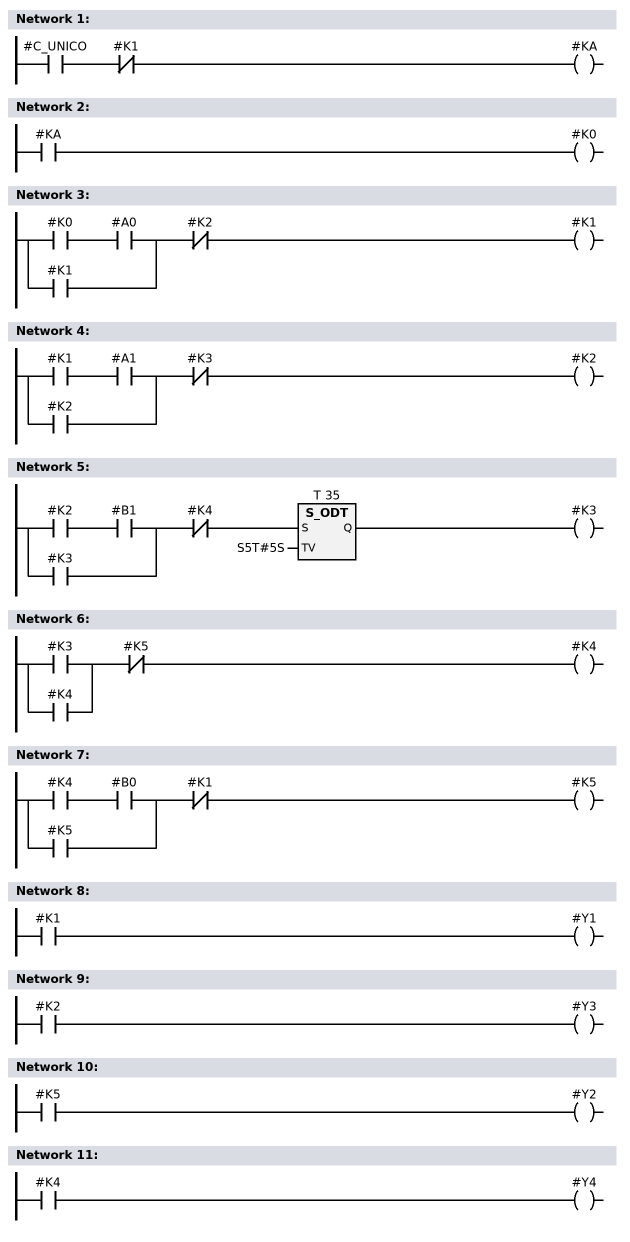
NETWORK
TITLE =
      A     #C_UNICO;
      AN    #K1;
      =     #KA;
NETWORK
TITLE =
      A     #KA;
      =     #K0;
NETWORK
TITLE =
      A(;
      A     #K0;
      A     #A0;
      O     #K1;
      );
      AN    #K2;
      =     #K1;
NETWORK
TITLE =
      A(;
      A     #K1;
      A     #A1;
      O     #K2;
      );
      AN    #K3;
      =     #K2;
NETWORK
TITLE =
      A(;
      A     #K2;
      A     #B1;
      O     #K3;
      );
      AN    #K4;
      L     S5T#5S;
      SD    T 35;
      NOP   0;
      NOP   0;
      NOP   0;
      A     T 35;
      =     #K3;
NETWORK
TITLE =
      A(;
      O     #K3;
      O     #K4;
      );
      AN    #K5;
      =     #K4;
NETWORK
TITLE =
      A(;
      A     #K4;
      A     #B0;
      O     #K5;
      );
      AN    #K1;
      =     #K5;
NETWORK
TITLE =
      A     #K1;
      =     #Y1;
NETWORK
TITLE =
      A     #K2;
      =     #Y3;
NETWORK
TITLE =
      A     #K5;
      =     #Y2;
NETWORK
TITLE =
      A     #K4;
      =     #Y4;
END_FUNCTION_BLOCK

FUNCTION_BLOCK "Ejercicio 6-3"	// FB 14
VERSION : 0.1
VAR_INPUT
  HONGO : BOOL ;
  RESET : BOOL ;
  C_UNICO : BOOL ;
  C_CONTINUO : BOOL ;
  PARO : BOOL ;
  DET_PIEZA : BOOL ;
  A0 : BOOL ;
  A1 : BOOL ;
  B0 : BOOL ;
  B1 : BOOL ;
  C0 : BOOL ;
  C1 : BOOL ;
END_VAR
VAR_OUTPUT
  Y1 : BOOL ;
  Y2 : BOOL ;
  Y3 : BOOL ;
  Y4 : BOOL ;
  Y5 : BOOL ;
  Y6 : BOOL ;
END_VAR
VAR
  K_PEM : BOOL ;
  KA : BOOL ;
  KB : BOOL ;
  K0 : BOOL ;
  K1 : BOOL ;
  K2 : BOOL ;
  K3 : BOOL ;
  K4 : BOOL ;
  K5 : BOOL ;
  K6 : BOOL ;
  K7 : BOOL ;
  K8 : BOOL ;
END_VAR
BEGIN
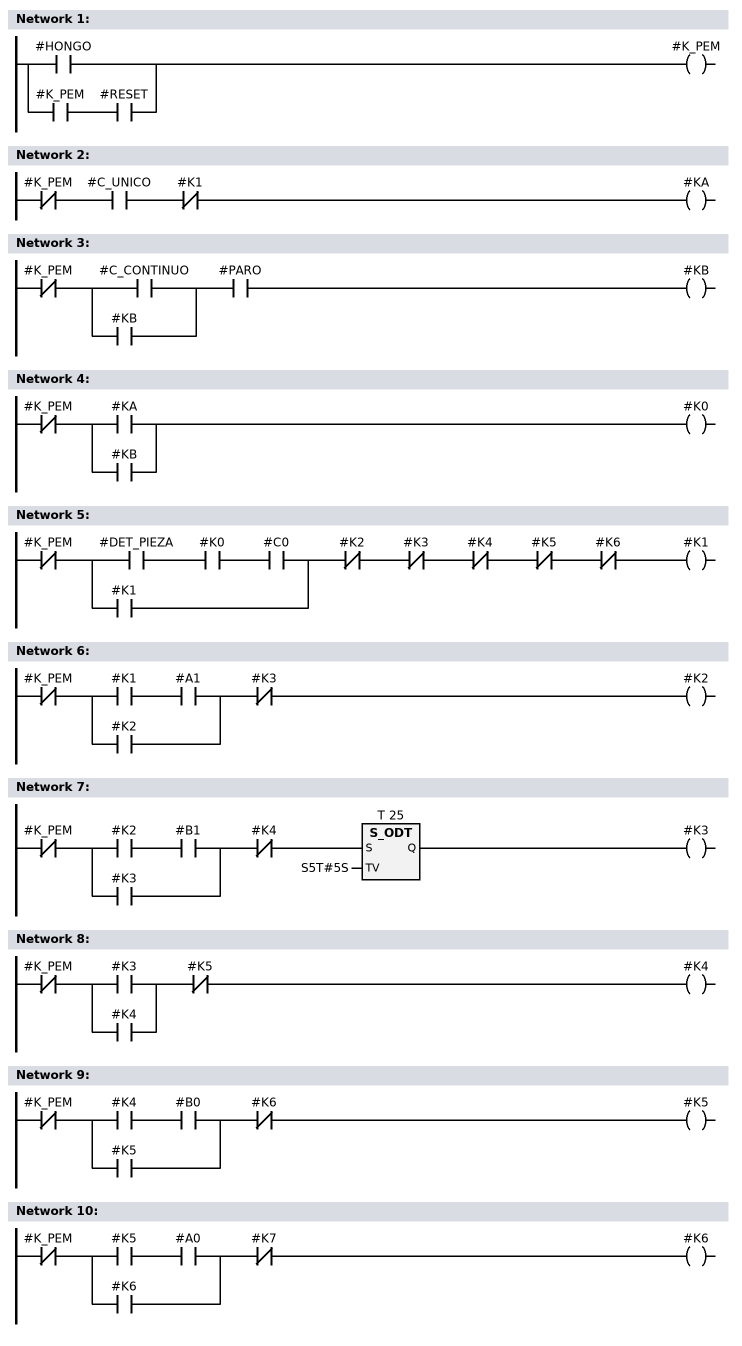
NETWORK
TITLE =
      O     #HONGO;
      O;
      A     #K_PEM;
      A     #RESET;
      =     #K_PEM;
NETWORK
TITLE =
      AN    #K_PEM;
      A     #C_UNICO;
      AN    #K1;
      =     #KA;
NETWORK
TITLE =
      AN    #K_PEM;
      A(;
      O     #C_CONTINUO;
      O     #KB;
      );
      A     #PARO;
      =     #KB;
NETWORK
TITLE =
      AN    #K_PEM;
      A(;
      O     #KA;
      O     #KB;
      );
      =     #K0;
NETWORK
TITLE =
      AN    #K_PEM;
      A(;
      A     #DET_PIEZA;
      A     #K0;
      A     #C0;
      O     #K1;
      );
      AN    #K2;
      AN    #K3;
      AN    #K4;
      AN    #K5;
      AN    #K6;
      =     #K1;
NETWORK
TITLE =
      AN    #K_PEM;
      A(;
      A     #K1;
      A     #A1;
      O     #K2;
      );
      AN    #K3;
      =     #K2;
NETWORK
TITLE =
      AN    #K_PEM;
      A(;
      A     #K2;
      A     #B1;
      O     #K3;
      );
      AN    #K4;
      L     S5T#5S;
      SD    T 25;
      NOP   0;
      NOP   0;
      NOP   0;
      A     T 25;
      =     #K3;
NETWORK
TITLE =
      AN    #K_PEM;
      A(;
      O     #K3;
      O     #K4;
      );
      AN    #K5;
      =     #K4;
NETWORK
TITLE =
      AN    #K_PEM;
      A(;
      A     #K4;
      A     #B0;
      O     #K5;
      );
      AN    #K6;
      =     #K5;
NETWORK
TITLE =
      AN    #K_PEM;
      A(;
      A     #K5;
      A     #A0;
      O     #K6;
      );
      AN    #K7;
      =     #K6;
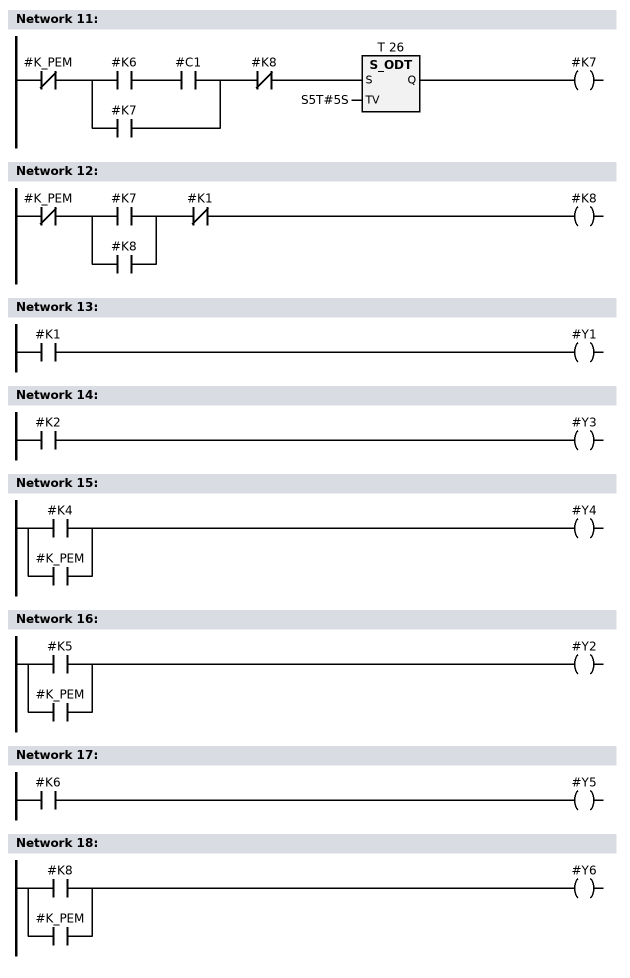
NETWORK
TITLE =
      AN    #K_PEM;
      A(;
      A     #K6;
      A     #C1;
      O     #K7;
      );
      AN    #K8;
      L     S5T#5S;
      SD    T 26;
      NOP   0;
      NOP   0;
      NOP   0;
      A     T 26;
      =     #K7;
NETWORK
TITLE =
      AN    #K_PEM;
      A(;
      O     #K7;
      O     #K8;
      );
      AN    #K1;
      =     #K8;
NETWORK
TITLE =
      A     #K1;
      =     #Y1;
NETWORK
TITLE =
      A     #K2;
      =     #Y3;
NETWORK
TITLE =
      O     #K4;
      O     #K_PEM;
      =     #Y4;
NETWORK
TITLE =
      O     #K5;
      O     #K_PEM;
      =     #Y2;
NETWORK
TITLE =
      A     #K6;
      =     #Y5;
NETWORK
TITLE =
      O     #K8;
      O     #K_PEM;
      =     #Y6;
END_FUNCTION_BLOCK

FUNCTION_BLOCK "Paro de emergencia"	// FB 99
VERSION : 0.1
VAR_INPUT
  HONGO : BOOL ;
  RESET : BOOL ;
END_VAR
VAR_OUTPUT
  K_PEM : BOOL ;
END_VAR
BEGIN
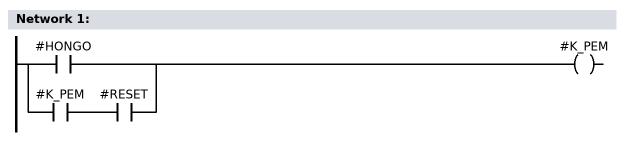
NETWORK
TITLE =
      O     #HONGO;
      O;
      A     #K_PEM;
      A     #RESET;
      =     #K_PEM;
END_FUNCTION_BLOCK

DATA_BLOCK DB 1
VERSION : 0.0
"Ejercicio1"
BEGIN
END_DATA_BLOCK

DATA_BLOCK DB 2
VERSION : 0.0
"Ejercicio 2"
BEGIN
END_DATA_BLOCK

DATA_BLOCK DB 3
VERSION : 0.0
"Ejercicio3"
BEGIN
END_DATA_BLOCK

DATA_BLOCK DB 4
VERSION : 0.0
"Ejercicio 4"
BEGIN
END_DATA_BLOCK

DATA_BLOCK DB 5
VERSION : 0.0
"Ejercicio 5"
BEGIN
END_DATA_BLOCK

DATA_BLOCK DB 6
VERSION : 0.0
"Ejercicio 6"
BEGIN
END_DATA_BLOCK

DATA_BLOCK DB 7
VERSION : 0.0
"Ejercicio C1"
BEGIN
END_DATA_BLOCK

DATA_BLOCK DB 8
VERSION : 0.0
"Ejercicio C2"
BEGIN
END_DATA_BLOCK

DATA_BLOCK DB 9
VERSION : 0.0
"Ejercicio 3-5"
BEGIN
END_DATA_BLOCK

DATA_BLOCK DB 10
VERSION : 0.0
"Ejercicio 3-6"
BEGIN
END_DATA_BLOCK

DATA_BLOCK DB 11
VERSION : 0.0
"Ejercicio 3-7"
BEGIN
END_DATA_BLOCK

DATA_BLOCK DB 12
VERSION : 0.0
"Ejercicio 6-1"
BEGIN
END_DATA_BLOCK

DATA_BLOCK DB 13
VERSION : 0.0
"Ejercicio 6-2"
BEGIN
END_DATA_BLOCK

DATA_BLOCK DB 14
VERSION : 0.0
"Ejercicio 6-3"
BEGIN
END_DATA_BLOCK

DATA_BLOCK DB 88
VERSION : 0.0
"Paro de emergencia"
BEGIN
END_DATA_BLOCK

DATA_BLOCK DB 89
VERSION : 0.0
"Paro de emergencia"
BEGIN
END_DATA_BLOCK

DATA_BLOCK DB 90
VERSION : 0.0
"Paro de emergencia"
BEGIN
END_DATA_BLOCK

DATA_BLOCK DB 91
VERSION : 0.0
"Paro de emergencia"
BEGIN
END_DATA_BLOCK

DATA_BLOCK DB 92
VERSION : 0.0
"Paro de emergencia"
BEGIN
END_DATA_BLOCK

DATA_BLOCK DB 93
VERSION : 0.0
"Paro de emergencia"
BEGIN
END_DATA_BLOCK

DATA_BLOCK DB 94
VERSION : 0.0
"Paro de emergencia"
BEGIN
END_DATA_BLOCK

DATA_BLOCK DB 95
VERSION : 0.0
"Paro de emergencia"
BEGIN
END_DATA_BLOCK

DATA_BLOCK DB 96
VERSION : 0.0
"Paro de emergencia"
BEGIN
END_DATA_BLOCK

DATA_BLOCK DB 97
VERSION : 0.0
"Paro de emergencia"
BEGIN
END_DATA_BLOCK

DATA_BLOCK DB 98
VERSION : 0.0
"Paro de emergencia"
BEGIN
END_DATA_BLOCK

DATA_BLOCK DB 99
VERSION : 0.0
"Paro de emergencia"
BEGIN
END_DATA_BLOCK

ORGANIZATION_BLOCK "CYCL_EXC"	// OB 1
TITLE = "Main Program Sweep (Cycle)"
VERSION : 0.1
VAR_TEMP
  OB1_EV_CLASS : BYTE ;	//Bits 0-3 = 1 (Coming event), Bits 4-7 = 1 (Event class 1)
  OB1_SCAN_1 : BYTE ;	//1 (Cold restart scan 1 of OB 1), 3 (Scan 2-n of OB 1)
  OB1_PRIORITY : BYTE ;	//Priority of OB Execution
  OB1_OB_NUMBR : BYTE ;	//1 (Organization block 1, OB1)
  OB1_RESERVED_1 : BYTE ;	//Reserved for system
  OB1_RESERVED_2 : BYTE ;	//Reserved for system
  OB1_PREV_CYCLE : INT ;	//Cycle time of previous OB1 scan (milliseconds)
  OB1_MIN_CYCLE : INT ;	//Minimum cycle time of OB1 (milliseconds)
  OB1_MAX_CYCLE : INT ;	//Maximum cycle time of OB1 (milliseconds)
  OB1_DATE_TIME : DATE_AND_TIME ;	//Date and time OB1 started
END_VAR
BEGIN
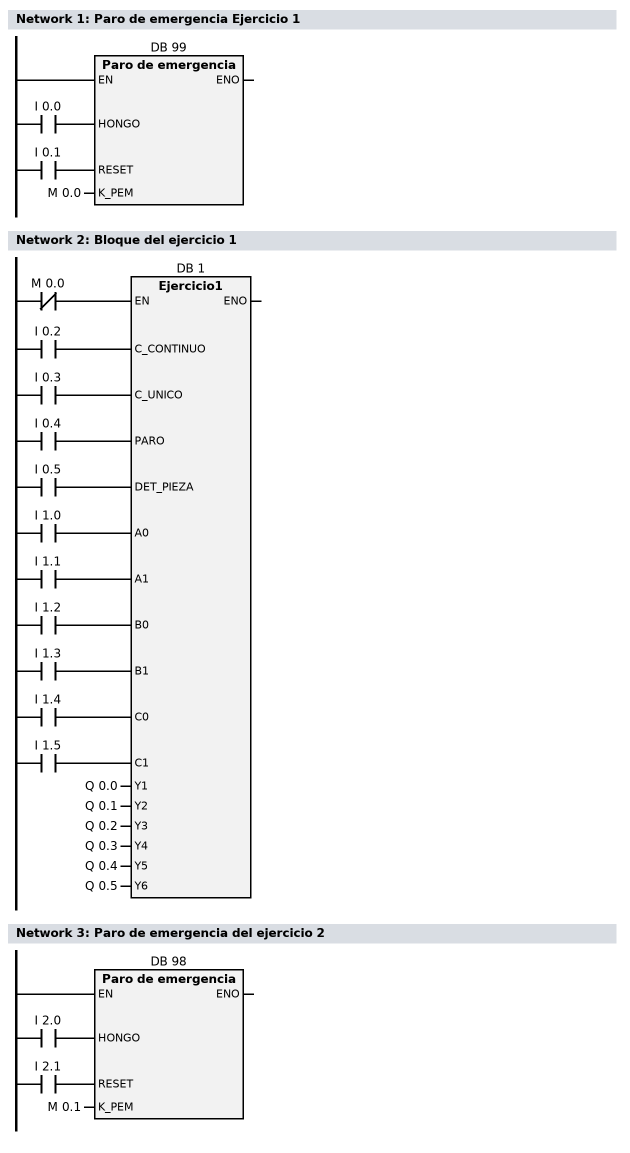
NETWORK
TITLE = Paro de emergencia Ejercicio 1
      A     I 0.0;
      =     L 20.0;
      BLD   103;
      A     I 0.1;
      =     L 20.1;
      BLD   103;
      CALL  "Paro de emergencia" , DB 99 (
           HONGO                    := L 20.0,
           RESET                    := L 20.1,
           K_PEM                    := M 0.0);
      NOP   0;
NETWORK
TITLE = Bloque del ejercicio 1
      A     I 0.2;
      =     L 20.0;
      BLD   103;
      A     I 0.3;
      =     L 20.1;
      BLD   103;
      A     I 0.4;
      =     L 20.2;
      BLD   103;
      A     I 0.5;
      =     L 20.3;
      BLD   103;
      A     I 1.0;
      =     L 20.4;
      BLD   103;
      A     I 1.1;
      =     L 20.5;
      BLD   103;
      A     I 1.2;
      =     L 20.6;
      BLD   103;
      A     I 1.3;
      =     L 20.7;
      BLD   103;
      A     I 1.4;
      =     L 21.0;
      BLD   103;
      A     I 1.5;
      =     L 21.1;
      BLD   103;
      AN    M 0.0;
      JNB   _001;
      CALL  "Ejercicio1" , DB 1 (
           C_CONTINUO               := L 20.0,
           C_UNICO                  := L 20.1,
           PARO                     := L 20.2,
           DET_PIEZA                := L 20.3,
           A0                       := L 20.4,
           A1                       := L 20.5,
           B0                       := L 20.6,
           B1                       := L 20.7,
           C0                       := L 21.0,
           C1                       := L 21.1,
           Y1                       := Q 0.0,
           Y2                       := Q 0.1,
           Y3                       := Q 0.2,
           Y4                       := Q 0.3,
           Y5                       := Q 0.4,
           Y6                       := Q 0.5);
_001: NOP   0;
NETWORK
TITLE = Paro de emergencia del ejercicio 2
      A     I 2.0;
      =     L 20.0;
      BLD   103;
      A     I 2.1;
      =     L 20.1;
      BLD   103;
      CALL  "Paro de emergencia" , DB 98 (
           HONGO                    := L 20.0,
           RESET                    := L 20.1,
           K_PEM                    := M 0.1);
      NOP   0;
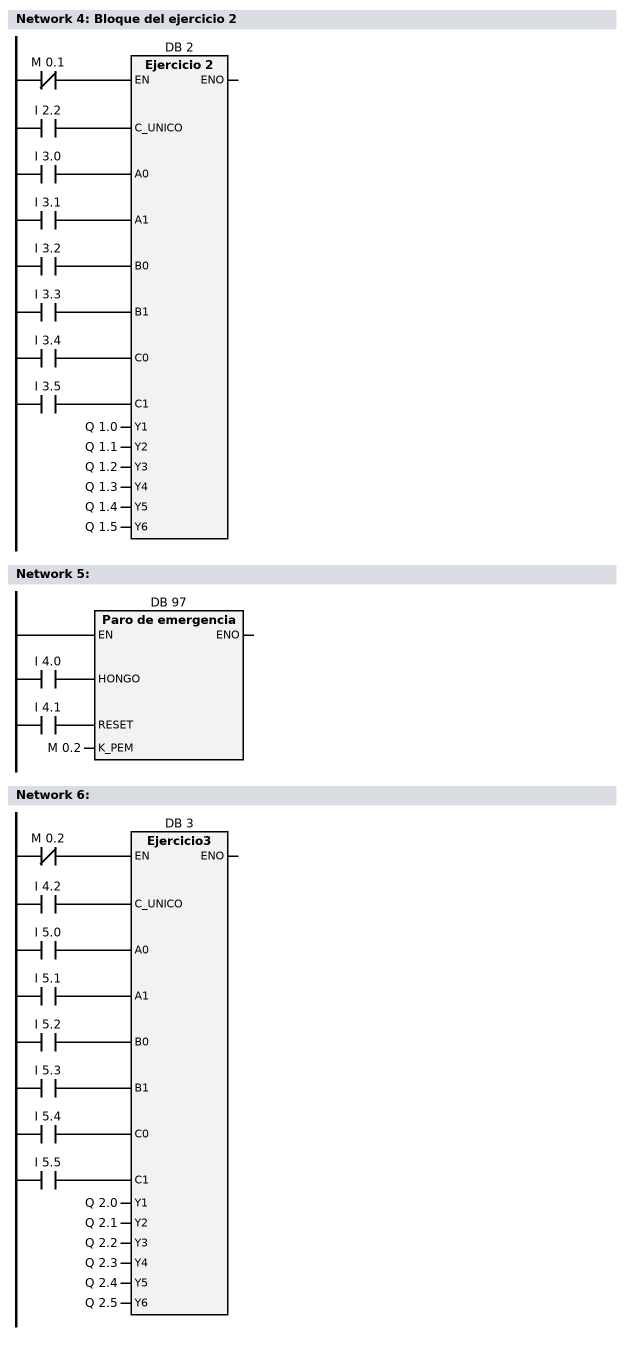
NETWORK
TITLE = Bloque del ejercicio 2
      A     I 2.2;
      =     L 20.0;
      BLD   103;
      A     I 3.0;
      =     L 20.1;
      BLD   103;
      A     I 3.1;
      =     L 20.2;
      BLD   103;
      A     I 3.2;
      =     L 20.3;
      BLD   103;
      A     I 3.3;
      =     L 20.4;
      BLD   103;
      A     I 3.4;
      =     L 20.5;
      BLD   103;
      A     I 3.5;
      =     L 20.6;
      BLD   103;
      AN    M 0.1;
      JNB   _002;
      CALL  "Ejercicio 2" , DB 2 (
           C_UNICO                  := L 20.0,
           A0                       := L 20.1,
           A1                       := L 20.2,
           B0                       := L 20.3,
           B1                       := L 20.4,
           C0                       := L 20.5,
           C1                       := L 20.6,
           Y1                       := Q 1.0,
           Y2                       := Q 1.1,
           Y3                       := Q 1.2,
           Y4                       := Q 1.3,
           Y5                       := Q 1.4,
           Y6                       := Q 1.5);
_002: NOP   0;
NETWORK
TITLE =
      A     I 4.0;
      =     L 20.0;
      BLD   103;
      A     I 4.1;
      =     L 20.1;
      BLD   103;
      CALL  "Paro de emergencia" , DB 97 (
           HONGO                    := L 20.0,
           RESET                    := L 20.1,
           K_PEM                    := M 0.2);
      NOP   0;
NETWORK
TITLE =
      A     I 4.2;
      =     L 20.0;
      BLD   103;
      A     I 5.0;
      =     L 20.1;
      BLD   103;
      A     I 5.1;
      =     L 20.2;
      BLD   103;
      A     I 5.2;
      =     L 20.3;
      BLD   103;
      A     I 5.3;
      =     L 20.4;
      BLD   103;
      A     I 5.4;
      =     L 20.5;
      BLD   103;
      A     I 5.5;
      =     L 20.6;
      BLD   103;
      AN    M 0.2;
      JNB   _003;
      CALL  "Ejercicio3" , DB 3 (
           C_UNICO                  := L 20.0,
           A0                       := L 20.1,
           A1                       := L 20.2,
           B0                       := L 20.3,
           B1                       := L 20.4,
           C0                       := L 20.5,
           C1                       := L 20.6,
           Y1                       := Q 2.0,
           Y2                       := Q 2.1,
           Y3                       := Q 2.2,
           Y4                       := Q 2.3,
           Y5                       := Q 2.4,
           Y6                       := Q 2.5);
_003: NOP   0;
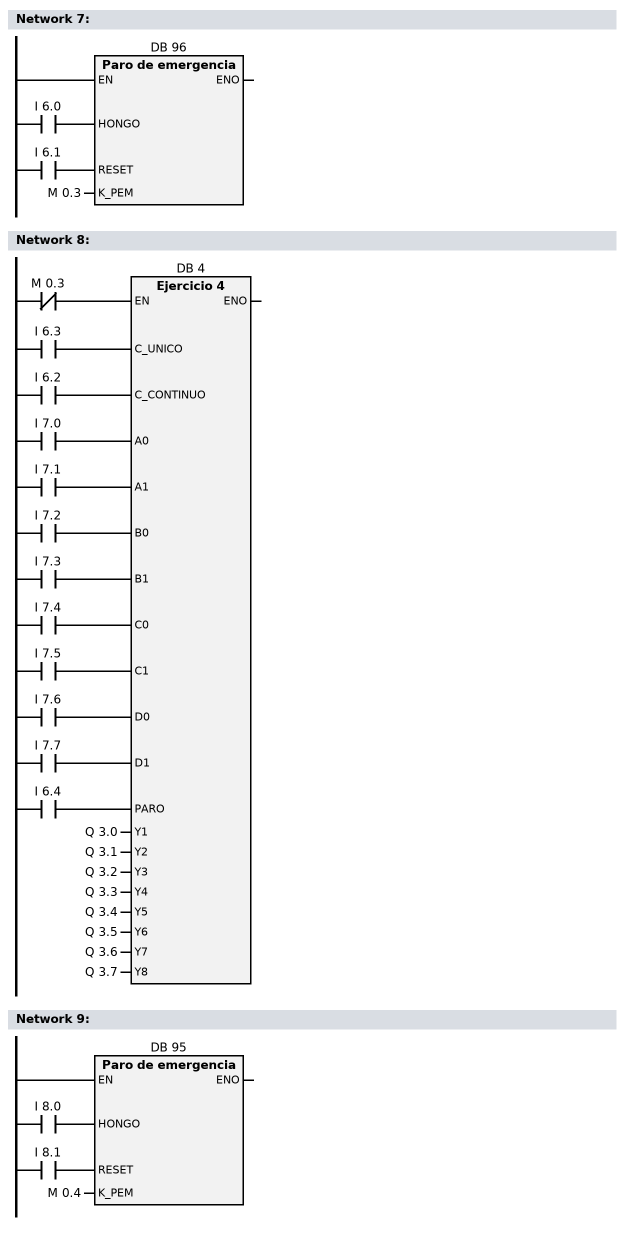
NETWORK
TITLE =
      A     I 6.0;
      =     L 20.0;
      BLD   103;
      A     I 6.1;
      =     L 20.1;
      BLD   103;
      CALL  "Paro de emergencia" , DB 96 (
           HONGO                    := L 20.0,
           RESET                    := L 20.1,
           K_PEM                    := M 0.3);
      NOP   0;
NETWORK
TITLE =
      A     I 6.3;
      =     L 20.0;
      BLD   103;
      A     I 6.2;
      =     L 20.1;
      BLD   103;
      A     I 7.0;
      =     L 20.2;
      BLD   103;
      A     I 7.1;
      =     L 20.3;
      BLD   103;
      A     I 7.2;
      =     L 20.4;
      BLD   103;
      A     I 7.3;
      =     L 20.5;
      BLD   103;
      A     I 7.4;
      =     L 20.6;
      BLD   103;
      A     I 7.5;
      =     L 20.7;
      BLD   103;
      A     I 7.6;
      =     L 21.0;
      BLD   103;
      A     I 7.7;
      =     L 21.1;
      BLD   103;
      A     I 6.4;
      =     L 21.2;
      BLD   103;
      AN    M 0.3;
      JNB   _004;
      CALL  "Ejercicio 4" , DB 4 (
           C_UNICO                  := L 20.0,
           C_CONTINUO               := L 20.1,
           A0                       := L 20.2,
           A1                       := L 20.3,
           B0                       := L 20.4,
           B1                       := L 20.5,
           C0                       := L 20.6,
           C1                       := L 20.7,
           D0                       := L 21.0,
           D1                       := L 21.1,
           PARO                     := L 21.2,
           Y1                       := Q 3.0,
           Y2                       := Q 3.1,
           Y3                       := Q 3.2,
           Y4                       := Q 3.3,
           Y5                       := Q 3.4,
           Y6                       := Q 3.5,
           Y7                       := Q 3.6,
           Y8                       := Q 3.7);
_004: NOP   0;
NETWORK
TITLE =
      A     I 8.0;
      =     L 20.0;
      BLD   103;
      A     I 8.1;
      =     L 20.1;
      BLD   103;
      CALL  "Paro de emergencia" , DB 95 (
           HONGO                    := L 20.0,
           RESET                    := L 20.1,
           K_PEM                    := M 0.4);
      NOP   0;
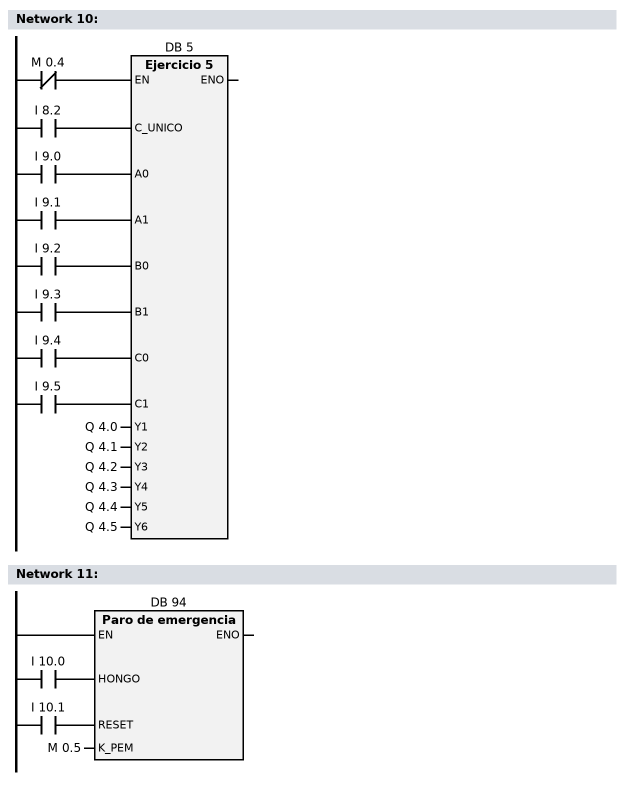
NETWORK
TITLE =
      A     I 8.2;
      =     L 20.0;
      BLD   103;
      A     I 9.0;
      =     L 20.1;
      BLD   103;
      A     I 9.1;
      =     L 20.2;
      BLD   103;
      A     I 9.2;
      =     L 20.3;
      BLD   103;
      A     I 9.3;
      =     L 20.4;
      BLD   103;
      A     I 9.4;
      =     L 20.5;
      BLD   103;
      A     I 9.5;
      =     L 20.6;
      BLD   103;
      AN    M 0.4;
      JNB   _005;
      CALL  "Ejercicio 5" , DB 5 (
           C_UNICO                  := L 20.0,
           A0                       := L 20.1,
           A1                       := L 20.2,
           B0                       := L 20.3,
           B1                       := L 20.4,
           C0                       := L 20.5,
           C1                       := L 20.6,
           Y1                       := Q 4.0,
           Y2                       := Q 4.1,
           Y3                       := Q 4.2,
           Y4                       := Q 4.3,
           Y5                       := Q 4.4,
           Y6                       := Q 4.5);
_005: NOP   0;
NETWORK
TITLE =
      A     I 10.0;
      =     L 20.0;
      BLD   103;
      A     I 10.1;
      =     L 20.1;
      BLD   103;
      CALL  "Paro de emergencia" , DB 94 (
           HONGO                    := L 20.0,
           RESET                    := L 20.1,
           K_PEM                    := M 0.5);
      NOP   0;
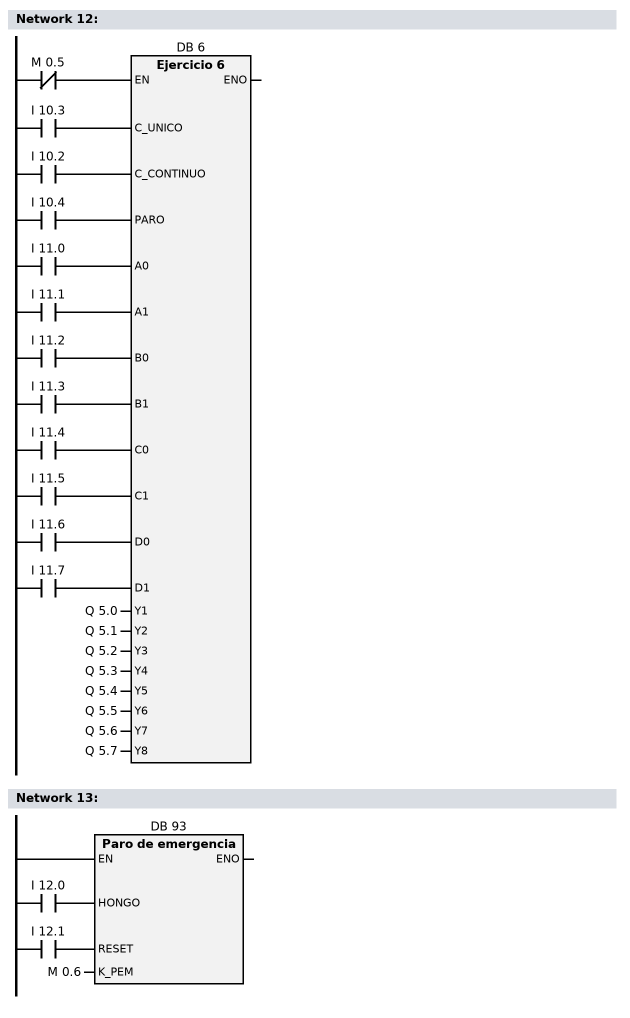
NETWORK
TITLE =
      A     I 10.3;
      =     L 20.0;
      BLD   103;
      A     I 10.2;
      =     L 20.1;
      BLD   103;
      A     I 10.4;
      =     L 20.2;
      BLD   103;
      A     I 11.0;
      =     L 20.3;
      BLD   103;
      A     I 11.1;
      =     L 20.4;
      BLD   103;
      A     I 11.2;
      =     L 20.5;
      BLD   103;
      A     I 11.3;
      =     L 20.6;
      BLD   103;
      A     I 11.4;
      =     L 20.7;
      BLD   103;
      A     I 11.5;
      =     L 21.0;
      BLD   103;
      A     I 11.6;
      =     L 21.1;
      BLD   103;
      A     I 11.7;
      =     L 21.2;
      BLD   103;
      AN    M 0.5;
      JNB   _006;
      CALL  "Ejercicio 6" , DB 6 (
           C_UNICO                  := L 20.0,
           C_CONTINUO               := L 20.1,
           PARO                     := L 20.2,
           A0                       := L 20.3,
           A1                       := L 20.4,
           B0                       := L 20.5,
           B1                       := L 20.6,
           C0                       := L 20.7,
           C1                       := L 21.0,
           D0                       := L 21.1,
           D1                       := L 21.2,
           Y1                       := Q 5.0,
           Y2                       := Q 5.1,
           Y3                       := Q 5.2,
           Y4                       := Q 5.3,
           Y5                       := Q 5.4,
           Y6                       := Q 5.5,
           Y7                       := Q 5.6,
           Y8                       := Q 5.7);
_006: NOP   0;
NETWORK
TITLE =
      A     I 12.0;
      =     L 20.0;
      BLD   103;
      A     I 12.1;
      =     L 20.1;
      BLD   103;
      CALL  "Paro de emergencia" , DB 93 (
           HONGO                    := L 20.0,
           RESET                    := L 20.1,
           K_PEM                    := M 0.6);
      NOP   0;
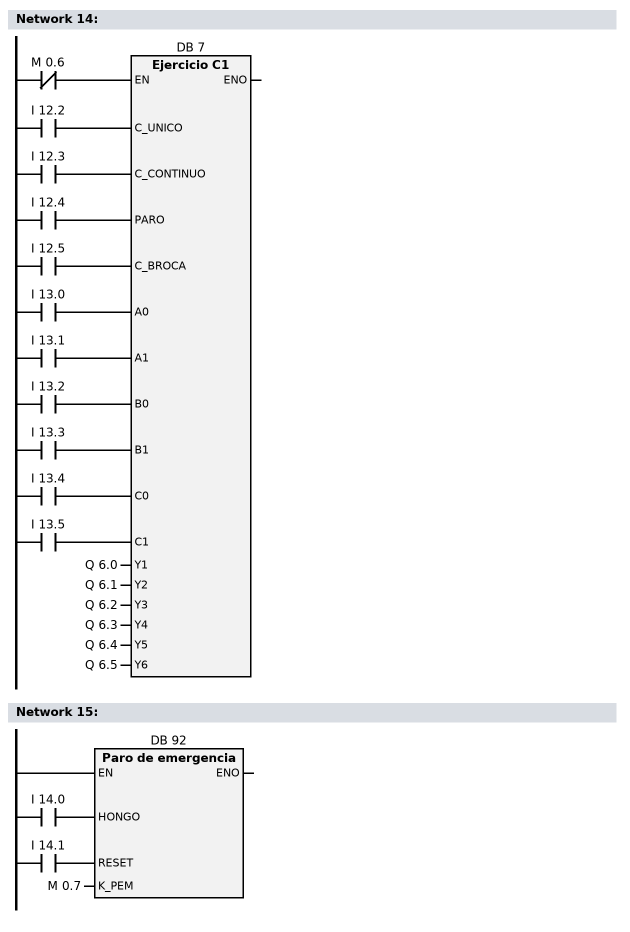
NETWORK
TITLE =
      A     I 12.2;
      =     L 20.0;
      BLD   103;
      A     I 12.3;
      =     L 20.1;
      BLD   103;
      A     I 12.4;
      =     L 20.2;
      BLD   103;
      A     I 12.5;
      =     L 20.3;
      BLD   103;
      A     I 13.0;
      =     L 20.4;
      BLD   103;
      A     I 13.1;
      =     L 20.5;
      BLD   103;
      A     I 13.2;
      =     L 20.6;
      BLD   103;
      A     I 13.3;
      =     L 20.7;
      BLD   103;
      A     I 13.4;
      =     L 21.0;
      BLD   103;
      A     I 13.5;
      =     L 21.1;
      BLD   103;
      AN    M 0.6;
      JNB   _007;
      CALL  "Ejercicio C1" , DB 7 (
           C_UNICO                  := L 20.0,
           C_CONTINUO               := L 20.1,
           PARO                     := L 20.2,
           C_BROCA                  := L 20.3,
           A0                       := L 20.4,
           A1                       := L 20.5,
           B0                       := L 20.6,
           B1                       := L 20.7,
           C0                       := L 21.0,
           C1                       := L 21.1,
           Y1                       := Q 6.0,
           Y2                       := Q 6.1,
           Y3                       := Q 6.2,
           Y4                       := Q 6.3,
           Y5                       := Q 6.4,
           Y6                       := Q 6.5);
_007: NOP   0;
NETWORK
TITLE =
      A     I 14.0;
      =     L 20.0;
      BLD   103;
      A     I 14.1;
      =     L 20.1;
      BLD   103;
      CALL  "Paro de emergencia" , DB 92 (
           HONGO                    := L 20.0,
           RESET                    := L 20.1,
           K_PEM                    := M 0.7);
      NOP   0;
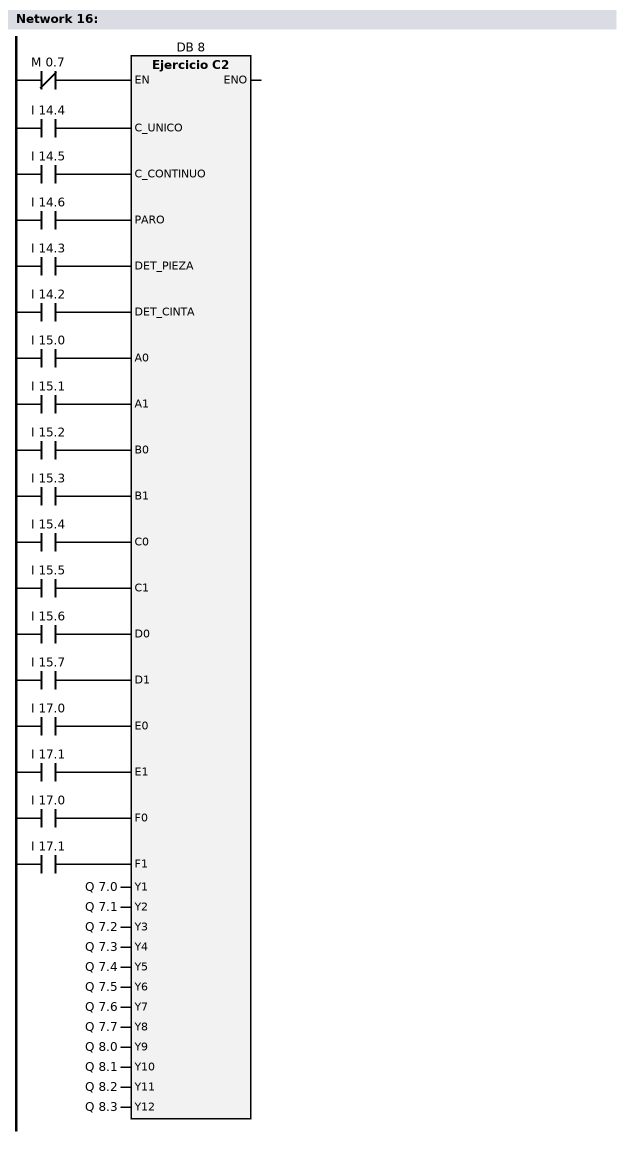
NETWORK
TITLE =
      A     I 14.4;
      =     L 20.0;
      BLD   103;
      A     I 14.5;
      =     L 20.1;
      BLD   103;
      A     I 14.6;
      =     L 20.2;
      BLD   103;
      A     I 14.3;
      =     L 20.3;
      BLD   103;
      A     I 14.2;
      =     L 20.4;
      BLD   103;
      A     I 15.0;
      =     L 20.5;
      BLD   103;
      A     I 15.1;
      =     L 20.6;
      BLD   103;
      A     I 15.2;
      =     L 20.7;
      BLD   103;
      A     I 15.3;
      =     L 21.0;
      BLD   103;
      A     I 15.4;
      =     L 21.1;
      BLD   103;
      A     I 15.5;
      =     L 21.2;
      BLD   103;
      A     I 15.6;
      =     L 21.3;
      BLD   103;
      A     I 15.7;
      =     L 21.4;
      BLD   103;
      A     I 17.0;
      =     L 21.5;
      BLD   103;
      A     I 17.1;
      =     L 21.6;
      BLD   103;
      A     I 17.0;
      =     L 21.7;
      BLD   103;
      A     I 17.1;
      =     L 22.0;
      BLD   103;
      AN    M 0.7;
      JNB   _008;
      CALL  "Ejercicio C2" , DB 8 (
           C_UNICO                  := L 20.0,
           C_CONTINUO               := L 20.1,
           PARO                     := L 20.2,
           DET_PIEZA                := L 20.3,
           DET_CINTA                := L 20.4,
           A0                       := L 20.5,
           A1                       := L 20.6,
           B0                       := L 20.7,
           B1                       := L 21.0,
           C0                       := L 21.1,
           C1                       := L 21.2,
           D0                       := L 21.3,
           D1                       := L 21.4,
           E0                       := L 21.5,
           E1                       := L 21.6,
           F0                       := L 21.7,
           F1                       := L 22.0,
           Y1                       := Q 7.0,
           Y2                       := Q 7.1,
           Y3                       := Q 7.2,
           Y4                       := Q 7.3,
           Y5                       := Q 7.4,
           Y6                       := Q 7.5,
           Y7                       := Q 7.6,
           Y8                       := Q 7.7,
           Y9                       := Q 8.0,
           Y10                      := Q 8.1,
           Y11                      := Q 8.2,
           Y12                      := Q 8.3);
_008: NOP   0;
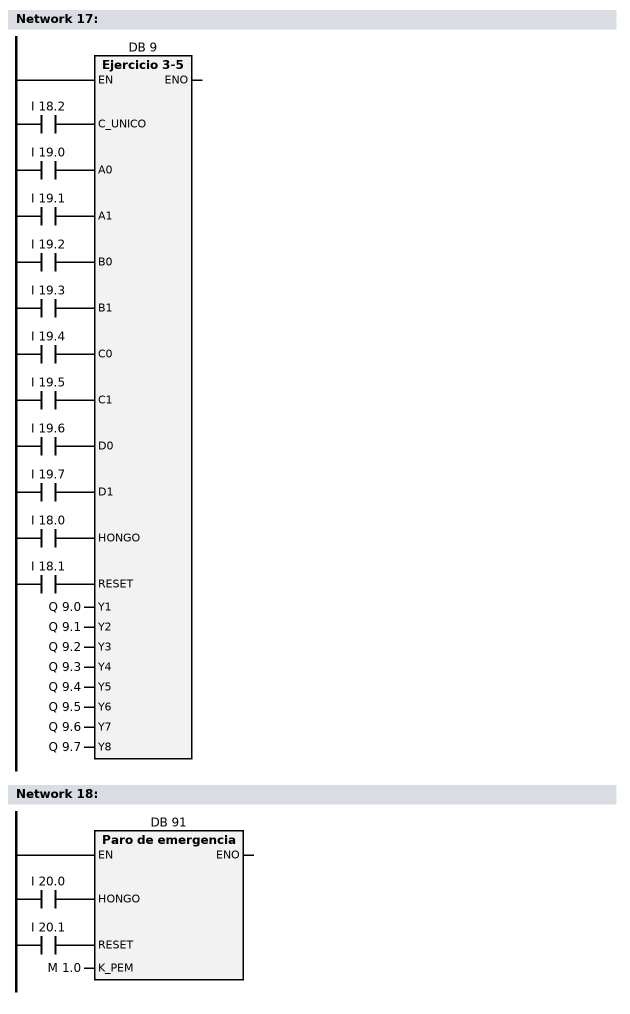
NETWORK
TITLE =
      A     I 18.2;
      =     L 20.0;
      BLD   103;
      A     I 19.0;
      =     L 20.1;
      BLD   103;
      A     I 19.1;
      =     L 20.2;
      BLD   103;
      A     I 19.2;
      =     L 20.3;
      BLD   103;
      A     I 19.3;
      =     L 20.4;
      BLD   103;
      A     I 19.4;
      =     L 20.5;
      BLD   103;
      A     I 19.5;
      =     L 20.6;
      BLD   103;
      A     I 19.6;
      =     L 20.7;
      BLD   103;
      A     I 19.7;
      =     L 21.0;
      BLD   103;
      A     I 18.0;
      =     L 21.1;
      BLD   103;
      A     I 18.1;
      =     L 21.2;
      BLD   103;
      CALL  "Ejercicio 3-5" , DB 9 (
           C_UNICO                  := L 20.0,
           A0                       := L 20.1,
           A1                       := L 20.2,
           B0                       := L 20.3,
           B1                       := L 20.4,
           C0                       := L 20.5,
           C1                       := L 20.6,
           D0                       := L 20.7,
           D1                       := L 21.0,
           HONGO                    := L 21.1,
           RESET                    := L 21.2,
           Y1                       := Q 9.0,
           Y2                       := Q 9.1,
           Y3                       := Q 9.2,
           Y4                       := Q 9.3,
           Y5                       := Q 9.4,
           Y6                       := Q 9.5,
           Y7                       := Q 9.6,
           Y8                       := Q 9.7);
      NOP   0;
NETWORK
TITLE =
      A     I 20.0;
      =     L 20.0;
      BLD   103;
      A     I 20.1;
      =     L 20.1;
      BLD   103;
      CALL  "Paro de emergencia" , DB 91 (
           HONGO                    := L 20.0,
           RESET                    := L 20.1,
           K_PEM                    := M 1.0);
      NOP   0;
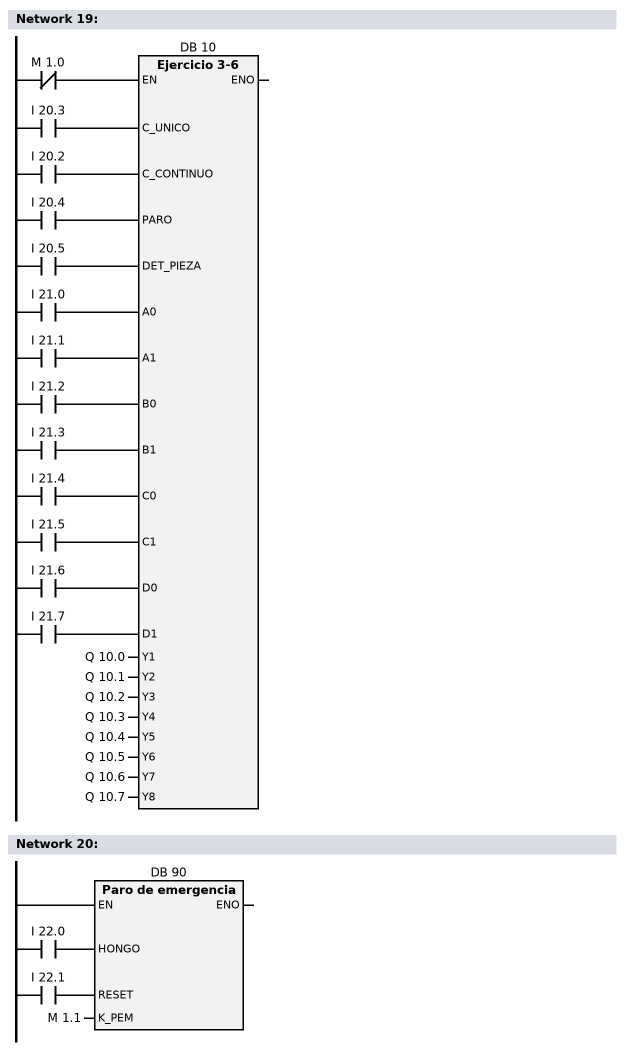
NETWORK
TITLE =
      A     I 20.3;
      =     L 20.0;
      BLD   103;
      A     I 20.2;
      =     L 20.1;
      BLD   103;
      A     I 20.4;
      =     L 20.2;
      BLD   103;
      A     I 20.5;
      =     L 20.3;
      BLD   103;
      A     I 21.0;
      =     L 20.4;
      BLD   103;
      A     I 21.1;
      =     L 20.5;
      BLD   103;
      A     I 21.2;
      =     L 20.6;
      BLD   103;
      A     I 21.3;
      =     L 20.7;
      BLD   103;
      A     I 21.4;
      =     L 21.0;
      BLD   103;
      A     I 21.5;
      =     L 21.1;
      BLD   103;
      A     I 21.6;
      =     L 21.2;
      BLD   103;
      A     I 21.7;
      =     L 21.3;
      BLD   103;
      AN    M 1.0;
      JNB   _009;
      CALL  "Ejercicio 3-6" , DB 10 (
           C_UNICO                  := L 20.0,
           C_CONTINUO               := L 20.1,
           PARO                     := L 20.2,
           DET_PIEZA                := L 20.3,
           A0                       := L 20.4,
           A1                       := L 20.5,
           B0                       := L 20.6,
           B1                       := L 20.7,
           C0                       := L 21.0,
           C1                       := L 21.1,
           D0                       := L 21.2,
           D1                       := L 21.3,
           Y1                       := Q 10.0,
           Y2                       := Q 10.1,
           Y3                       := Q 10.2,
           Y4                       := Q 10.3,
           Y5                       := Q 10.4,
           Y6                       := Q 10.5,
           Y7                       := Q 10.6,
           Y8                       := Q 10.7);
_009: NOP   0;
NETWORK
TITLE =
      A     I 22.0;
      =     L 20.0;
      BLD   103;
      A     I 22.1;
      =     L 20.1;
      BLD   103;
      CALL  "Paro de emergencia" , DB 90 (
           HONGO                    := L 20.0,
           RESET                    := L 20.1,
           K_PEM                    := M 1.1);
      NOP   0;
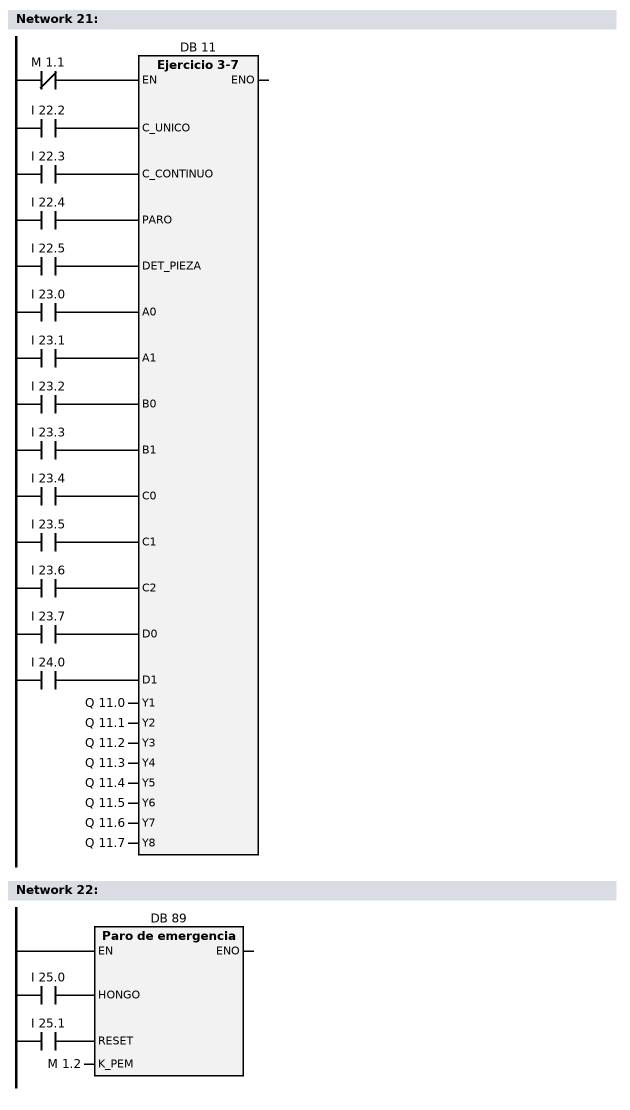
NETWORK
TITLE =
      A     I 22.2;
      =     L 20.0;
      BLD   103;
      A     I 22.3;
      =     L 20.1;
      BLD   103;
      A     I 22.4;
      =     L 20.2;
      BLD   103;
      A     I 22.5;
      =     L 20.3;
      BLD   103;
      A     I 23.0;
      =     L 20.4;
      BLD   103;
      A     I 23.1;
      =     L 20.5;
      BLD   103;
      A     I 23.2;
      =     L 20.6;
      BLD   103;
      A     I 23.3;
      =     L 20.7;
      BLD   103;
      A     I 23.4;
      =     L 21.0;
      BLD   103;
      A     I 23.5;
      =     L 21.1;
      BLD   103;
      A     I 23.6;
      =     L 21.2;
      BLD   103;
      A     I 23.7;
      =     L 21.3;
      BLD   103;
      A     I 24.0;
      =     L 21.4;
      BLD   103;
      AN    M 1.1;
      JNB   _00a;
      CALL  "Ejercicio 3-7" , DB 11 (
           C_UNICO                  := L 20.0,
           C_CONTINUO               := L 20.1,
           PARO                     := L 20.2,
           DET_PIEZA                := L 20.3,
           A0                       := L 20.4,
           A1                       := L 20.5,
           B0                       := L 20.6,
           B1                       := L 20.7,
           C0                       := L 21.0,
           C1                       := L 21.1,
           C2                       := L 21.2,
           D0                       := L 21.3,
           D1                       := L 21.4,
           Y1                       := Q 11.0,
           Y2                       := Q 11.1,
           Y3                       := Q 11.2,
           Y4                       := Q 11.3,
           Y5                       := Q 11.4,
           Y6                       := Q 11.5,
           Y7                       := Q 11.6,
           Y8                       := Q 11.7);
_00a: NOP   0;
NETWORK
TITLE =
      A     I 25.0;
      =     L 20.0;
      BLD   103;
      A     I 25.1;
      =     L 20.1;
      BLD   103;
      CALL  "Paro de emergencia" , DB 89 (
           HONGO                    := L 20.0,
           RESET                    := L 20.1,
           K_PEM                    := M 1.2);
      NOP   0;
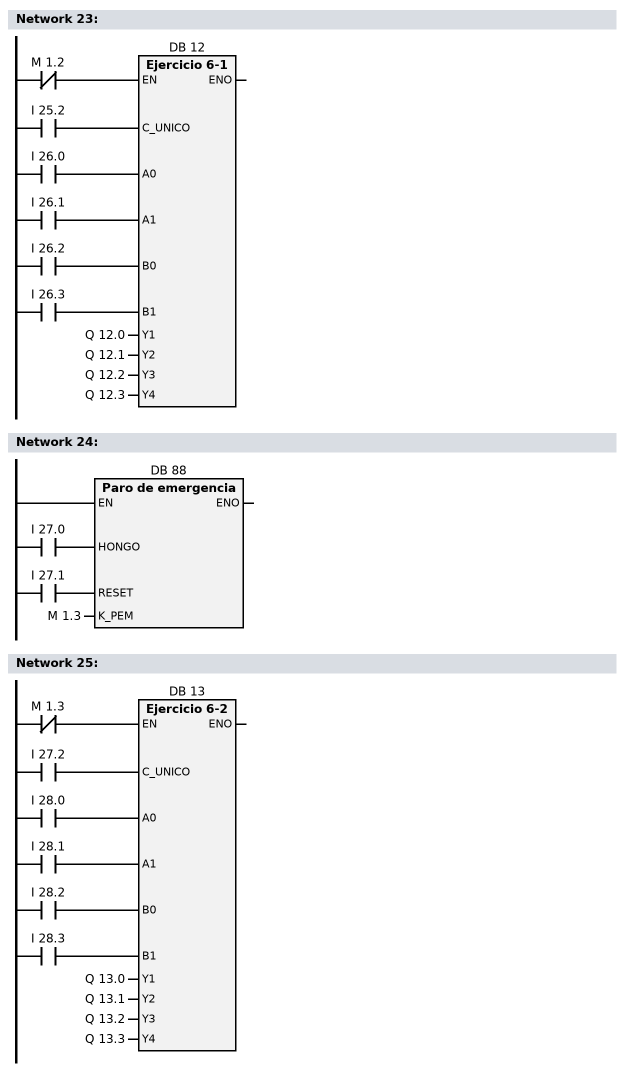
NETWORK
TITLE =
      A     I 25.2;
      =     L 20.0;
      BLD   103;
      A     I 26.0;
      =     L 20.1;
      BLD   103;
      A     I 26.1;
      =     L 20.2;
      BLD   103;
      A     I 26.2;
      =     L 20.3;
      BLD   103;
      A     I 26.3;
      =     L 20.4;
      BLD   103;
      AN    M 1.2;
      JNB   _00b;
      CALL  "Ejercicio 6-1" , DB 12 (
           C_UNICO                  := L 20.0,
           A0                       := L 20.1,
           A1                       := L 20.2,
           B0                       := L 20.3,
           B1                       := L 20.4,
           Y1                       := Q 12.0,
           Y2                       := Q 12.1,
           Y3                       := Q 12.2,
           Y4                       := Q 12.3);
_00b: NOP   0;
NETWORK
TITLE =
      A     I 27.0;
      =     L 20.0;
      BLD   103;
      A     I 27.1;
      =     L 20.1;
      BLD   103;
      CALL  "Paro de emergencia" , DB 88 (
           HONGO                    := L 20.0,
           RESET                    := L 20.1,
           K_PEM                    := M 1.3);
      NOP   0;
NETWORK
TITLE =
      A     I 27.2;
      =     L 20.0;
      BLD   103;
      A     I 28.0;
      =     L 20.1;
      BLD   103;
      A     I 28.1;
      =     L 20.2;
      BLD   103;
      A     I 28.2;
      =     L 20.3;
      BLD   103;
      A     I 28.3;
      =     L 20.4;
      BLD   103;
      AN    M 1.3;
      JNB   _00c;
      CALL  "Ejercicio 6-2" , DB 13 (
           C_UNICO                  := L 20.0,
           A0                       := L 20.1,
           A1                       := L 20.2,
           B0                       := L 20.3,
           B1                       := L 20.4,
           Y1                       := Q 13.0,
           Y2                       := Q 13.1,
           Y3                       := Q 13.2,
           Y4                       := Q 13.3);
_00c: NOP   0;
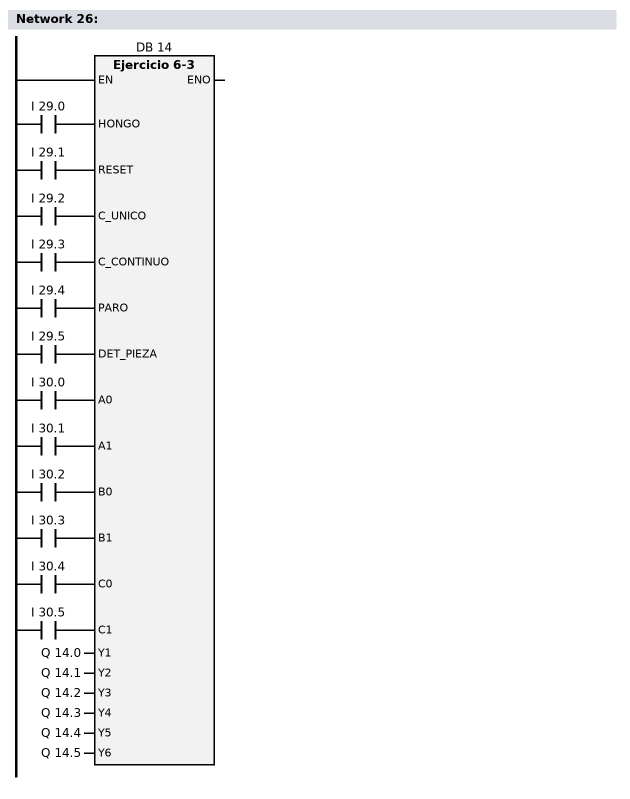
NETWORK
TITLE =
      A     I 29.0;
      =     L 20.0;
      BLD   103;
      A     I 29.1;
      =     L 20.1;
      BLD   103;
      A     I 29.2;
      =     L 20.2;
      BLD   103;
      A     I 29.3;
      =     L 20.3;
      BLD   103;
      A     I 29.4;
      =     L 20.4;
      BLD   103;
      A     I 29.5;
      =     L 20.5;
      BLD   103;
      A     I 30.0;
      =     L 20.6;
      BLD   103;
      A     I 30.1;
      =     L 20.7;
      BLD   103;
      A     I 30.2;
      =     L 21.0;
      BLD   103;
      A     I 30.3;
      =     L 21.1;
      BLD   103;
      A     I 30.4;
      =     L 21.2;
      BLD   103;
      A     I 30.5;
      =     L 21.3;
      BLD   103;
      CALL  "Ejercicio 6-3" , DB 14 (
           HONGO                    := L 20.0,
           RESET                    := L 20.1,
           C_UNICO                  := L 20.2,
           C_CONTINUO               := L 20.3,
           PARO                     := L 20.4,
           DET_PIEZA                := L 20.5,
           A0                       := L 20.6,
           A1                       := L 20.7,
           B0                       := L 21.0,
           B1                       := L 21.1,
           C0                       := L 21.2,
           C1                       := L 21.3,
           Y1                       := Q 14.0,
           Y2                       := Q 14.1,
           Y3                       := Q 14.2,
           Y4                       := Q 14.3,
           Y5                       := Q 14.4,
           Y6                       := Q 14.5);
      NOP   0;
END_ORGANIZATION_BLOCK
